INTERFACE ITF_DEV_AnaIn

END_INTERFACE

(* stored: Version 1.1.0.1, ProductVersion 3.1.4024.12
   Itf ITF_DEV_AnaIn: Id {de2eb338-209c-4dd0-bbf6-2a45293efce7} *)
